// TIA Portal V17 export
// export: Created 2021-12-03T08:13:13.1192243Z, ExportSetting WithDefaults, DisplayName Totally Integrated Automation Portal, DisplayVersion V17, DisplayName TIA Portal Openness, DisplayVersion V17, DisplayName TIA Portal Version Control Interface, DisplayVersion V17, DisplayName STEP 7 Professional, DisplayVersion V17, DisplayName STEP 7 Safety, DisplayVersion V17, DisplayName WinCC Advanced, DisplayVersion V17
DATA_BLOCK "FDBI_Safety_Perimeter"   // DB301, F_DB
VERSION : 0.1
// stored: AutoNumber false, InstanceOfName FFB_Safety_Perimeter, InstanceOfType FB
"FFB_Safety_Perimeter"
   // VAR_INPUT
   //    I_ReqAckCls : Bool;
   //    I_PrDrCls : Bool;
   //    I_ReqCnfrm : Bool;
   //    I_SpRdyOpn : Bool;
   //    I_AckFltRst : Bool;
   //    I_EmrStp : Bool;
   //    I_KeyConv : Bool;
   //    I_SPBreak : Bool;
   // END_VAR
   // VAR_OUTPUT
   //    O_SPClose : Bool;
   //    O_RdySPCls_P3 : Bool;
   //    O_AckSPCls : Bool;
   //    O_OpnP : Bool;
   //    O_SPBreak : Bool;
   // END_VAR
   // VAR
   //    S_AckSPClsP3_SR : Bool;
   //    S_AckSPClsP3_HIS : Bool;
   //    S_AckSPRst_TON { S7_SetPoint := 'True'} : TON;
   //    S_SP_Close_SR : Bool;
   //    S_AckSPClsP_HIS : Bool;
   //    S_SPBreak_SR : Bool;
   //    S_AckSPOpn_TON { S7_SetPoint := 'True'} : TON;
   //    S_AckSPOpn_SR : Bool;
   //    S_AckSPOpnP_HIS : Bool;
   // END_VAR
BEGIN
END_DATA_BLOCK
